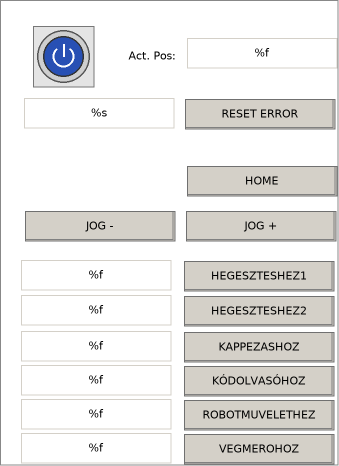
VISUALIZATION TempPistiTengely  // 339x466
    PowerSwitch (22,26 83x61), variable: GVL.bPistiServo, behaviour: TOGGLE, style: Switch-PowerSwitch-Blue
    Button (187,166 150x30), "HOME"
        OnMouseUp: execute { PISTITENGELY.sPistiAxisCommand:='HOME'; }
    Button (186,211 150x30), "JOG +"
        tap PISTITENGELY.bPistiJOGPlus
    Button (25,211 150x30), "JOG -"
        tap PISTITENGELY.bPistiJOGMinus
    Button (185,99 150x30), "RESET ERROR"
        tap PISTITENGELY.bPistiReset
    Textfield (24,98 150x30), "%s", text variable: PISTITENGELY.nPistiErrorCode, input disabled if: TRUE
    Textfield (21,260 150x30), "%f", text variable: GVL.lrHegesztoPosition6
        OnMouseClick: write the text variable via VisuDialogs.Numpad, min -10000, max -1
    Button (184,261 150x30), "HEGESZTESHEZ1"
        OnMouseUp: execute { PISTITENGELY.lrPistiPosition:=GVL.lrHegesztoPosition6; PISTITENGELY.sPistiAxisCommand:='MOVE'; }
    Label (77,41 150x30), "Act. Pos:"
    Textfield (187,38 150x30), "%f", text variable: PISTITENGELY.lrPistiActPos, input disabled if: TRUE
    Textfield (21,331 150x30), "%f", text variable: GVL.lrKappePosition
        OnMouseClick: write the text variable via VisuDialogs.Numpad, min -10000, max -1
    Button (184,332 150x30), "KAPPEZASHOZ"
        OnMouseUp: execute { PISTITENGELY.lrPistiPosition:=GVL.lrKappePosition; PISTITENGELY.sPistiAxisCommand:='MOVE'; }
    Textfield (21,399 150x30), "%f", text variable: GVL.lrRobotKappePosition
        OnMouseClick: write the text variable via VisuDialogs.Numpad, min -10000, max -1
    Button (184,400 150x30), "ROBOTMUVELETHEZ"
        OnMouseUp: execute { PISTITENGELY.lrPistiPosition:=GVL.lrRobotKappePosition; PISTITENGELY.sPistiAxisCommand:='MOVE'; }
    Textfield (21,433 150x30), "%f", text variable: GVL.lrVegmeroPosition
        OnMouseClick: write the text variable via VisuDialogs.Numpad, min -10000, max -1
    Button (184,434 150x30), "VEGMEROHOZ"
        OnMouseUp: execute { PISTITENGELY.lrPistiPosition:=GVL.lrVegmeroPosition; PISTITENGELY.sPistiAxisCommand:='MOVE'; }
    Textfield (21,295 150x30), "%f", text variable: GVL.lrHegesztoPosition7
        OnMouseClick: write the text variable via VisuDialogs.Numpad, min -10000, max -1
    Button (184,296 150x30), "HEGESZTESHEZ2"
        OnMouseUp: execute { PISTITENGELY.lrPistiPosition:=GVL.lrHegesztoPosition7; PISTITENGELY.sPistiAxisCommand:='MOVE'; }
    Textfield (21,365 150x30), "%f", text variable: GVL.lrKodolvasasPosition
        OnMouseClick: write the text variable via VisuDialogs.Numpad, min -10000, max -1
    Button (184,366 150x30), "KÓDOLVASÓHOZ"
        OnMouseUp: execute { PISTITENGELY.lrPistiPosition:=GVL.lrKodolvasasPosition; PISTITENGELY.sPistiAxisCommand:='MOVE'; }
END_VISUALIZATION

(* stored: Version 1.1.0.1, ProductVersion 3.1.4024.11
   Visu TempPistiTengely: Id {5a999ad2-b0da-46d4-9c69-cce46b7d26cb} *)
